{attribute 'linkalways'} 
{attribute 'no_explicit_call' := 'This FB is a CLASS and must be accessed using methods or properties'}
{attribute 'enable_dynamic_creation'}
FUNCTION_BLOCK _BOOL EXTENDS DatatypeBase
VAR
	localData : BOOL;
	activeData : REFERENCE TO BOOL REF= localData;
END_VAR

PROPERTY PUBLIC Address : PVOID
GET
Address := ADR(activeData);
END_GET
END_PROPERTY

METHOD PUBLIC ClearReference
VAR_INPUT
END_VAR
activeData REF= localData;
END_METHOD

METHOD PUBLIC Clone : I_Datatype
VAR
    pClone : POINTER TO _BOOL;
END_VAR
pClone := __NEW(_BOOL(InitialValue := Value));
Clone := pClone^;
END_METHOD

METHOD FB_init : BOOL
VAR_INPUT
	bInitRetains : BOOL; // if TRUE, the retain variables are initialized (warm start / cold start)
	bInCopyCode : BOOL;  // if TRUE, the instance afterwards gets moved into the copy code (online change)
	InitialValue : BOOL;
END_VAR
localData := InitialValue;
END_METHOD

PROPERTY PUBLIC Identifier : T_MAXSTRING
GET
Identifier := 'BOOL';
END_GET
END_PROPERTY

METHOD PUBLIC SerializeTypeWith
VAR_INPUT
	Serializer : I_Serializer;
END_VAR
Serializer.StartObject();
Serializer.AddKeyString('type','BOOL');
Serializer.EndObject();
END_METHOD

METHOD PUBLIC SerializeWith
VAR_INPUT
	Serializer : I_Serializer;
END_VAR
Serializer.AddBool(activeData);
END_METHOD

PROPERTY PUBLIC Size : UDINT
GET
Size := SIZEOF(activeData);
END_GET
END_PROPERTY

METHOD TryDeserializeFrom : BOOL
VAR_INPUT
	Deserializer : I_Deserializer;
END_VAR
TryDeserializeFrom := Deserializer.TryGetBool(activeData);
END_METHOD

METHOD TryMakeReferenceOf : BOOL
VAR_INPUT
	Target : I_Datatype;
END_VAR
VAR
	pTargetData : POINTER TO BOOL;
END_VAR
IF NOT (Target.Identifier = Identifier) THEN
	RETURN;
END_IF

pTargetData := Target.Address;
activeData REF= pTargetData^;
TryMakeReferenceOf := TRUE;
END_METHOD

PROPERTY PUBLIC Value : BOOL
GET
Value := activeData;
END_GET
SET
activeData := Value;
END_SET
END_PROPERTY

END_FUNCTION_BLOCK

(* stored: Version 1.1.0.1, ProductVersion 3.1.4024.12
   POU _BOOL: Id {73f2c26e-32e9-46f5-a312-2927d449c86e}, SpecialFunc None
   Folder Constructor: Id {39988db6-a8a1-475d-94a6-59b54070f4c4}
   Property Address: Id {4148f607-b9df-4d1a-bf8e-18043a110c15}
   Get Get: Id {456d7a9f-e62e-4265-b148-685ad336bdb8}
   Method ClearReference: Id {2c9e366f-88fb-029e-3dc8-beea96060188}
   Method Clone: Id {a0f61c7d-9075-49a5-ae2f-6fa56ea65ce9}
   Method FB_init: Id {b9c2f4cc-3d64-49ec-b0f9-94f6b91f63cf}
   Property Identifier: Id {72af1979-c8a6-44ae-8e4c-a01801501cf1}
   Get Get: Id {3733e778-83b4-4688-aec0-b56df0af7a48}
   Method SerializeTypeWith: Id {713b8a57-0816-4acb-80e0-2d0e5c479dc0}
   Method SerializeWith: Id {0c38b446-0e15-4d4f-ad5d-632b1b0e0167}
   Property Size: Id {b7f8d582-eff3-4ad7-b504-ea24c9d0588e}
   Get Get: Id {0cded36b-91a1-4cad-b4de-a6bed829e204}
   Method TryDeserializeFrom: Id {a78fdf0d-71c4-4c7c-8b8a-311686fb692b}
   Method TryMakeReferenceOf: Id {7005b362-8e83-054d-2624-d6bbb82e7b1c}
   Property Value: Id {c45fd22d-2330-40b4-b235-05bd28ec9ac2}
   Get Get: Id {a72ad693-3f18-4a62-84e1-00ad91e8acdd}
   Set Set: Id {27a77381-a71a-4ebc-98ab-bbd5cc9c7e44} *)
